(* PLC project Unresolved reference, react-plc-diagram Invalid fixture 0.1.0 *)
(* stored: creationDateTime 2026-08-12T00:00:00Z, modificationDateTime 2026-08-12T00:00:00Z *)

PROGRAM BrokenReference

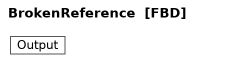
(* FBD diagram, written out as Structured Text *)
END_PROGRAM
